RoboDK station: VUI_control.rdk

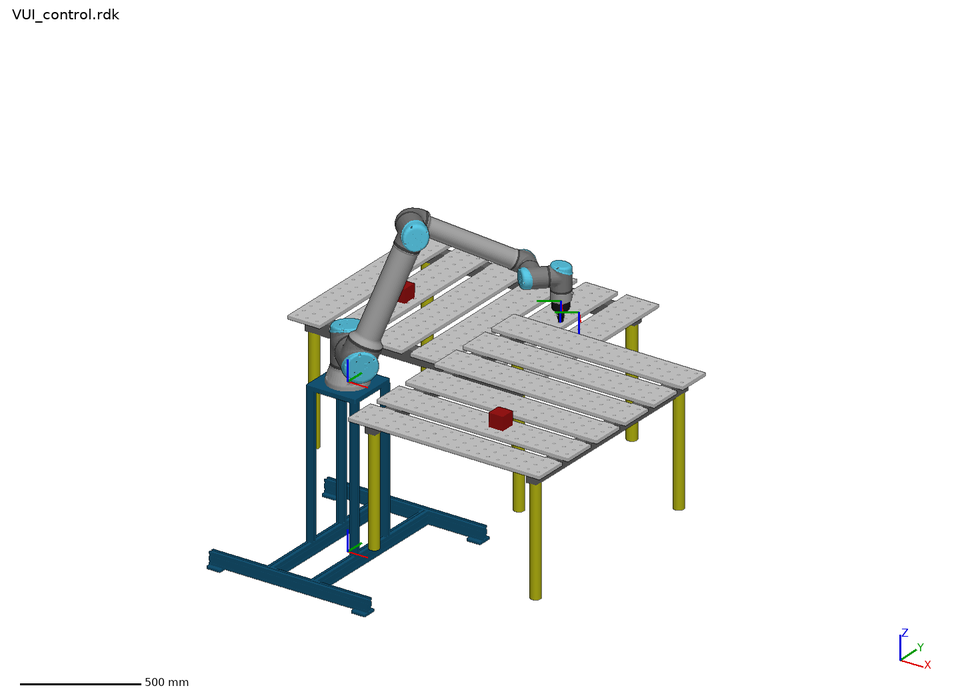
[picture v0: the station drawn from its stored meshes, robots at their saved joint values, targets as dots, program paths as lines]
Station Gripper_test (saved by RoboDK 5.3.1). Poses are relative to the parent item; angles as X-Y-Z fixed-axis rotations.
  - frame UR10e Base at (0, 0, 0) mm
    - robot UR10e: 6 axes, payload 10 kg, reach 1300 mm, repeatability 0.05 mm, weight 28.9 kg
        modified DH rows (alpha deg, a mm, theta deg, d mm): 0, 0, 0, 180.7; 90, 0, 180, 0; 0, 612.6, 0, 0; 0, 571.335, 0, 174.15; -90, 0, 0, 119.85; 90, 0, 180, 116.55
        joint limits [-360, -360, -360, -360, -360, -360] to [360, 360, 360, 360, 360, 360]; home [0, -90, -90, 0, 90, 0]; saved at [47.371, -112.765, -94.763, -63.434, 90.01, 8.604]
      - tool 2F85+FTS, TCP at (0, 0, 145) mm
      - frame RobotiQ 2F85 Base at (0, 0, 0) mm
        - robot RobotiQ 2F85: 1 axes, payload 5 kg
            joint limits [0] to [85]; home [85]; saved at [85]
        - target Open (Cartesian target) at (0, 0, 103.92) mm; joints [85] of RobotiQ 2F85
        - target Close (Cartesian target) at (0, 0, 103.92) mm; joints [3.08] of RobotiQ 2F85
        - frame ZED2i at (-64.91, -81.57, 83.4) mm
    - object Base-Robot at (0, 0, 0) mm, size 800 x 900 x 790 mm, geometry from Base-Robot.stl
  - Python program gripper_robotiq (listed below)
  - Python program main (listed below)
  - Python program UR_ActivateMonitoring (listed below)
  - frame Floor at (0, 0, -780) mm
    - object Pick_Table at (900, 0, 970) mm, rotated rx 0 ry 0 rz 90 deg, size 1193.8 x 965.2 x 609.6 mm, geometry from Object Table.wrl
      - object box at (-300, -80, 30) mm, size 71.9 x 71.9 x 71.9 mm, geometry from box.sld
    - object Place_Table at (0, 900, 750) mm, size 1193.8 x 965.2 x 609.6 mm, geometry from Object Table.wrl
      - object red at (-300, -80, 30) mm, size 71.9 x 71.9 x 71.9 mm, geometry from box.sld

--- Python program gripper_robotiq ---
"""Module to control Robotiq's grippers - tested with HAND-E"""

import socket
import threading
import time
from enum import Enum
from typing import Union, Tuple, OrderedDict


class RobotiqGripper:
    """
    Communicates with the gripper directly, via socket with string commands, leveraging string names for variables.
    """
    # WRITE VARIABLES (CAN ALSO READ)
    # act : activate (1 while activated, can be reset to clear fault status)
    ACT = 'ACT'
    # gto : go to (will perform go to with the actions set in pos, for, spe)
    GTO = 'GTO'
    ATR = 'ATR'  # atr : auto-release (emergency slow move)
    # adr : auto-release direction (open(1) or close(0) during auto-release)
    ADR = 'ADR'
    FOR = 'FOR'  # for : force (0-255)
    SPE = 'SPE'  # spe : speed (0-255)
    POS = 'POS'  # pos : position (0-255), 0 = open
    # READ VARIABLES
    STA = 'STA'  # status (0 = is reset, 1 = activating, 3 = active)
    PRE = 'PRE'  # position request (echo of last commanded position)
    # object detection (0 = moving, 1 = outer grip, 2 = inner grip, 3 = no object at rest)
    OBJ = 'OBJ'
    FLT = 'FLT'  # fault (0=ok, see manual for errors if not zero)

    ENCODING = 'UTF-8'  # ASCII and UTF-8 both seem to work

    class GripperStatus(Enum):
        """Gripper status reported by the gripper. The integer values have to match what the gripper sends."""
        RESET = 0
        ACTIVATING = 1
        # UNUSED = 2  # This value is currently not used by the gripper firmware
        ACTIVE = 3

    class ObjectStatus(Enum):
        """Object status reported by the gripper. The integer values have to match what the gripper sends."""
        MOVING = 0
        STOPPED_OUTER_OBJECT = 1
        STOPPED_INNER_OBJECT = 2
        AT_DEST = 3

    def __init__(self):
        """Constructor."""
        self.socket = None
        self.command_lock = threading.Lock()
        self._min_position = 0
        self._max_position = 255
        self._min_speed = 0
        self._max_speed = 255
        self._min_force = 0
        self._max_force = 255

    def connect(self, hostname: str, port: int, socket_timeout: float = 2.0) -> None:
        """Connects to a gripper at the given address.
        :param hostname: Hostname or ip.
        :param port: Port.
        :param socket_timeout: Timeout for blocking socket operations.
        """
        self.socket = socket.socket(socket.AF_INET, socket.SOCK_STREAM)
        self.socket.connect((hostname, port))
        self.socket.settimeout(socket_timeout)

    def disconnect(self) -> None:
        """Closes the connection with the gripper."""
        self.socket.close()

    def _set_vars(self, var_dict: OrderedDict[str, Union[int, float]]):
        """Sends the appropriate command via socket to set the value of n variables, and waits for its 'ack' response.
        :param var_dict: Dictionary of variables to set (variable_name, value).
        :return: True on successful reception of ack, false if no ack was received, indicating the set may not
        have been effective.
        """
        # construct unique command
        cmd = "SET"
        for variable, value in var_dict.items():
            cmd += f" {variable} {str(value)}"
        cmd += '\n'  # new line is required for the command to finish
        # atomic commands send/rcv
        with self.command_lock:
            self.socket.sendall(cmd.encode(self.ENCODING))
            data = self.socket.recv(1024)
        return self._is_ack(data)

    def _set_var(self, variable: str, value: Union[int, float]):
        """Sends the appropriate command via socket to set the value of a variable, and waits for its 'ack' response.
        :param variable: Variable to set.
        :param value: Value to set for the variable.
        :return: True on successful reception of ack, false if no ack was received, indicating the set may not
        have been effective.
        """
        return self._set_vars(OrderedDict([(variable, value)]))

    def _get_var(self, variable: str):
        """Sends the appropriate command to retrieve the value of a variable from the gripper, blocking until the
        response is received or the socket times out.
        :param variable: Name of the variable to retrieve.
        :return: Value of the variable as integer.
        """
        # atomic commands send/rcv
        with self.command_lock:
            cmd = f"GET {variable}\n"
            self.socket.sendall(cmd.encode(self.ENCODING))
            data = self.socket.recv(1024)

        # expect data of the form 'VAR x', where VAR is an echo of the variable name, and X the value
        # note some special variables (like FLT) may send 2 bytes, instead of an integer. We assume integer here
        var_name, value_str = data.decode(self.ENCODING).split()
        if var_name != variable:
            raise ValueError(
                f"Unexpected response {data} ({data.decode(self.ENCODING)}): does not match '{variable}'")
        value = int(value_str)
        return value

    @staticmethod
    def _is_ack(data: str):
        return data == b'ack'

    def _reset(self):
        """
        Reset the gripper.
        The following code is executed in the corresponding script function
        def rq_reset(gripper_socket="1"):
            rq_set_var("ACT", 0, gripper_socket)
            rq_set_var("ATR", 0, gripper_socket)

            while(not rq_get_var("ACT", 1, gripper_socket) == 0 or not rq_get_var("STA", 1, gripper_socket) == 0):
                rq_set_var("ACT", 0, gripper_socket)
                rq_set_var("ATR", 0, gripper_socket)
                sync()
            end

            sleep(0.5)
        end
        """
        self._set_var(self.ACT, 0)
        self._set_var(self.ATR, 0)
        while (not self._get_var(self.ACT) == 0 or not self._get_var(self.STA) == 0):
            self._set_var(self.ACT, 0)
            self._set_var(self.ATR, 0)
        time.sleep(0.5)

    def activate(self, auto_calibrate: bool = True):
        """Resets the activation flag in the gripper, and sets it back to one, clearing previous fault flags.
        :param auto_calibrate: Whether to calibrate the minimum and maximum positions based on actual motion.
        The following code is executed in the corresponding script function
        def rq_activate(gripper_socket="1"):
            if (not rq_is_gripper_activated(gripper_socket)):
                rq_reset(gripper_socket)

                while(not rq_get_var("ACT", 1, gripper_socket) == 0 or not rq_get_var("STA", 1, gripper_socket) == 0):
                    rq_reset(gripper_socket)
                    sync()
                end

                rq_set_var("ACT",1, gripper_socket)
            end
        end
        def rq_activate_and_wait(gripper_socket="1"):
            if (not rq_is_gripper_activated(gripper_socket)):
                rq_activate(gripper_socket)
                sleep(1.0)

                while(not rq_get_var("ACT", 1, gripper_socket) == 1 or not rq_get_var("STA", 1, gripper_socket) == 3):
                    sleep(0.1)
                end

                sleep(0.5)
            end
        end
        """
        if not self.is_active():
            self._reset()
            while (not self._get_var(self.ACT) == 0 or not self._get_var(self.STA) == 0):
                time.sleep(0.01)

            self._set_var(self.ACT, 1)
            time.sleep(1.0)
            while (not self._get_var(self.ACT) == 1 or not self._get_var(self.STA) == 3):
                time.sleep(0.01)

        # auto-calibrate position range if desired
        if auto_calibrate:
            self.auto_calibrate()

    def is_active(self):
        """Returns whether the gripper is active."""
        status = self._get_var(self.STA)
        return RobotiqGripper.GripperStatus(status) == RobotiqGripper.GripperStatus.ACTIVE

    def get_min_position(self) -> int:
        """Returns the minimum position the gripper can reach (open position)."""
        return self._min_position

    def get_max_position(self) -> int:
        """Returns the maximum position the gripper can reach (closed position)."""
        return self._max_position

    def get_open_position(self) -> int:
        """Returns what is considered the open position for gripper (minimum position value)."""
        return self.get_min_position()

    def get_closed_position(self) -> int:
        """Returns what is considered the closed position for gripper (maximum position value)."""
        return self.get_max_position()

    def is_open(self):
        """Returns whether the current position is considered as being fully open."""
        return self.get_current_position() <= self.get_open_position()

    def is_closed(self):
        """Returns whether the current position is considered as being fully closed."""
        return self.get_current_position() >= self.get_closed_position()

    def get_current_position(self) -> int:
        """Returns the current position as returned by the physical hardware."""
        return self._get_var(self.POS)

    def auto_calibrate(self, log: bool = True) -> None:
        """Attempts to calibrate the open and closed positions, by slowly closing and opening the gripper.
        :param log: Whether to print the results to log.
        """
        # first try to open in case we are holding an object
        (position, status) = self.move_and_wait_for_pos(
            self.get_open_position(), 64, 1)
        if RobotiqGripper.ObjectStatus(status) != RobotiqGripper.ObjectStatus.AT_DEST:
            raise RuntimeError(
                f"Calibration failed opening to start: {str(status)}")

        # try to close as far as possible, and record the number
        (position, status) = self.move_and_wait_for_pos(
            self.get_closed_position(), 64, 1)
        if RobotiqGripper.ObjectStatus(status) != RobotiqGripper.ObjectStatus.AT_DEST:
            raise RuntimeError(
                f"Calibration failed because of an object: {str(status)}")
        assert position <= self._max_position
        self._max_position = position

        # try to open as far as possible, and record the number
        (position, status) = self.move_and_wait_for_pos(
            self.get_open_position(), 64, 1)
        if RobotiqGripper.ObjectStatus(status) != RobotiqGripper.ObjectStatus.AT_DEST:
            raise RuntimeError(
                f"Calibration failed because of an object: {str(status)}")
        assert position >= self._min_position
        self._min_position = position

        if log:
            print(
                f"Gripper auto-calibrated to [{self.get_min_position()}, {self.get_max_position()}]")

    def move(self, position: int, speed: int, force: int) -> Tuple[bool, int]:
        """Sends commands to start moving towards the given position, with the specified speed and force.
        :param position: Position to move to [min_position, max_position]
        :param speed: Speed to move at [min_speed, max_speed]
        :param force: Force to use [min_force, max_force]
        :return: A tuple with a bool indicating whether the action it was successfully sent, and an integer with
        the actual position that was requested, after being adjusted to the min/max calibrated range.
        """

        def clip_val(min_val, val, max_val):
            return max(min_val, min(val, max_val))

        clip_pos = clip_val(self._min_position, position, self._max_position)
        clip_spe = clip_val(self._min_speed, speed, self._max_speed)
        clip_for = clip_val(self._min_force, force, self._max_force)

        # moves to the given position with the given speed and force
        var_dict = OrderedDict(
            [(self.POS, clip_pos), (self.SPE, clip_spe), (self.FOR, clip_for), (self.GTO, 1)])
        return self._set_vars(var_dict), clip_pos

    def move_and_wait_for_pos(self, position: int, speed: int, force: int) -> Tuple[int, ObjectStatus]:  # noqa
        """Sends commands to start moving towards the given position, with the specified speed and force, and
        then waits for the move to complete.
        :param position: Position to move to [min_position, max_position]
        :param speed: Speed to move at [min_speed, max_speed]
        :param force: Force to use [min_force, max_force]
        :return: A tuple with an integer representing the last position returned by the gripper after it notified
        that the move had completed, a status indicating how the move ended (see ObjectStatus enum for details). Note
        that it is possible that the position was not reached, if an object was detected during motion.
        """
        set_ok, cmd_pos = self.move(position, speed, force)
        if not set_ok:
            raise RuntimeError("Failed to set variables for move.")

        # wait until the gripper acknowledges that it will try to go to the requested position
        while self._get_var(self.PRE) != cmd_pos:
            time.sleep(0.001)

        # wait until not moving
        cur_obj = self._get_var(self.OBJ)
        while RobotiqGripper.ObjectStatus(cur_obj) == RobotiqGripper.ObjectStatus.MOVING:
            cur_obj = self._get_var(self.OBJ)

        # report the actual position and the object status
        final_pos = self._get_var(self.POS)
        final_obj = cur_obj
        return final_pos, RobotiqGripper.ObjectStatus(final_obj)

--- Python program main ---
try:  # 192.168.56.101
    from robodk.robolink import *
    from robodk import *
except:
    from robolink.robolink import *    # API to communicate with RoboDK
    from robodk.robodk import *      # basic matrix operations
finally:
    from AWSIoTPythonSDK.MQTTLib import AWSIoTMQTTClient
    import gripper_robotiq
    import socket
    import numpy as np
    import time
    import json
    import ast

    robot_ip = "192.168.1.10"  # Replace with your robot ip
    rdk_ip = 'localhost'  # Or the explicit ip of the computer running RoboDK
    pose = eye()

    RDK = Robolink()
    RDK.setRunMode(RUNMODE_RUN_ROBOT)  # RUNMODE_RUN_ROBOT
    robot = RDK.Item('UR10e')
    sim_gripper = RDK.Item('RobotiQ 2F85')  # the robotiq gripper inside RoboDK
    close_grp = RDK.Item("Close", ITEM_TYPE_TARGET)
    open_grp = RDK.Item("Open", ITEM_TYPE_TARGET)

    # detections=detector.GetData()

    gripper = gripper_robotiq.RobotiqGripper()
    gripper.connect(robot_ip, 63352)  # The port on the URe family is 63352
    # gripper.activate()
    gMax_Pos = gripper.get_max_position()

    clientId = "LAGID"
    host = "a1uv83ra8k1y7l-ats.iot.us-east-1.amazonaws.com"
    port = 8883
    rootCAPath = "C:/Users/LAG/Desktop/connect_device_package/root-CA.crt"
    privateKeyPath = "C:/Users/LAG/Desktop/connect_device_package/UR10_robot.private.key"
    certificatePath = "C:/Users/LAG/Desktop/connect_device_package/UR10_robot.cert.pem"
    topic_sub = "alexa/to/ur"
    topic_pub = "ur/to/alexa"
    mode = 'both'

    myAWSIoTMQTTClient = AWSIoTMQTTClient(clientId)  # ,useWebsocket=True)
    myAWSIoTMQTTClient.configureEndpoint(host, port)
    myAWSIoTMQTTClient.configureCredentials(
        rootCAPath, privateKeyPath, certificatePath)

    myAWSIoTMQTTClient.configureAutoReconnectBackoffTime(1, 32, 20)
    myAWSIoTMQTTClient.configureOfflinePublishQueueing(-1)
    myAWSIoTMQTTClient.configureDrainingFrequency(2)  # Draining: 2 Hz
    myAWSIoTMQTTClient.configureConnectDisconnectTimeout(10)  # 10 sec
    myAWSIoTMQTTClient.configureMQTTOperationTimeout(5)  # 5 sec
    myAWSIoTMQTTClient.connect()

    client_socket = socket.socket(socket.AF_INET, socket.SOCK_STREAM)
    host_ip = "10.25.147.84"
    port = 50007
    client_socket.connect((host_ip, port))

    # Global variables
    command_action = 0
    extra_value = 0
    name_save = ""
    current_prog = ""
    flag_create = False
    flag_frame = True
    flag_firstpoint = True
    gripper_status = True
    save_value = 0
    save_name = ""
    pick_flag = False
    place_flag = False

    state_record = 0
    speed = 150
    force = 20

    place_zone = [270, -90, 90, -90, -90, 0, False]
    pick_zone = [0, -90, -90, -90, 90, 0, True]

    class State(dict):
        def __setitem__(self, name, value):
            super().__setitem__(name, value)

    class Program:
        def __init__(self, home, frame, states):
            self.home = home
            self.frame = frame
            self.states = states

    def log_info(gripper):
        print(f"Pos: {str(gripper.get_current_position()): >3} "
              f"Open: {gripper.is_open(): <2} "
              f"Closed: {gripper.is_closed(): <2} ")

    def dt_gripper_position(current_position):
        dt_pos = [0]
        dt_pos[0] = 85 - (current_position / gMax_Pos) * 85
        return dt_pos

    def open_gripper():
        if RDK.RunMode() > 1:
            RDK.setRunMode(1)
        time.sleep(0.5)
        gripper.move_and_wait_for_pos(0, 255, 255)
        log_info(gripper)
        dt_pos = dt_gripper_position(gripper.get_current_position())
        sim_gripper.MoveJ(dt_pos)
        time.sleep(0.5)
        # tool_frame.DetachAll()
        RDK.setRunMode(6)
        time.sleep(0.5)

    def close_gripper():
        if RDK.RunMode() > 1:
            RDK.setRunMode(1)
        gripper.move_and_wait_for_pos(int(gMax_Pos/2), 255, 191)
        log_info(gripper)
        dt_pos = dt_gripper_position(gripper.get_current_position())
        sim_gripper.MoveJ(dt_pos)
        #input("Press 'Enter' to continue...")
        gripper.move_and_wait_for_pos(gMax_Pos, 255, 191)
        log_info(gripper)
        dt_pos = dt_gripper_position(gripper.get_current_position())
        sim_gripper.MoveJ(dt_pos)
        #input("Press 'Enter' to continue...")
        time.sleep(0.5)
        # tool_frame.AttachClosest()
        RDK.setRunMode(6)
        time.sleep(0.5)

    def publishMqtt(alert):
        # print("publishsing...")
        mess = {}
        mess["value"] = "mqtt"
        mess['message'] = alert
        messageJson = json.dumps(mess)
        myAWSIoTMQTTClient.publish(topic_pub, messageJson, 1)
        return 0

    def controlRobot(target):  # change when run or simulate
        global gripper_status
        if isinstance(target, list):
            robot.MoveJ(target)
            if target[6] == True:
                # sim_gripper.MoveJ(open_grp)
                gripper.move_and_wait_for_pos(5, speed, force)
                gripper_status = True
            else:
                # sim_gripper.MoveJ(close_grp)
                gripper.move_and_wait_for_pos(200, speed, force)
                gripper_status = False
        elif isinstance(target, dict):
            c = target.popitem()
            count = int(c[1])
            while count != 0:
                keys_list = [*target]  # list(target.keys())
                for key in keys_list:
                    robot.MoveJ(target[key])
                    if target[key][6] == True:
                        # sim_gripper.MoveJ(open_grp)
                        gripper.move_and_wait_for_pos(5, speed, force)
                    else:
                        # sim_gripper.MoveJ(close_grp)
                        gripper.move_and_wait_for_pos(200, speed, force)
                count -= 1
        elif target:
            gripper.move_and_wait_for_pos(target, speed, force)
            # sim_gripper.MoveJ(target)

        else:
            return 0

    def createProg(prog_name):
        with open("C:/Users/LAG/Documents/RoboDK/savedprog_data.json", "r") as jsonFile:
            savedPrograms = json.load(jsonFile)
        if prog_name in savedPrograms:
            return "A program with that name already exists, do you want to edit it? or try another name"
        else:
            global flag_create
            global current_prog
            flag_create = True
            prog = Program(None, None, State())
            savedPrograms[prog_name] = prog.__dict__
            with open("C:/Users/LAG/Documents/RoboDK/savedprog_data.json", "w") as jsonFile:
                json.dump(savedPrograms, jsonFile)
            jsonFile.close()
            current_prog = prog_name
            return f"{prog_name} was created succesfully"

    def selectFrame(frame):
        global flag_frame

        if flag_create == True or current_prog:
            with open('default_data.json', "r") as jsonFile:
                data = json.load(jsonFile)
                frame = data["frames"][frame]
            jsonFile.close()
            with open("C:/Users/LAG/Documents/RoboDK/savedprog_data.json", "r") as jsonFile:
                savedPrograms = json.load(jsonFile)
                savedPrograms[current_prog]["frame"] = frame
            with open("C:/Users/LAG/Documents/RoboDK/savedprog_data.json", "w") as jsonFile:
                json.dump(savedPrograms, jsonFile)
            jsonFile.close()
            flag_frame = True
            return "Frame saved succesfully"
        else:
            return "I need a program name"

    def selectFirstPoint(first_point):
        global flag_firstpoint
        if flag_create == True and flag_frame == True or current_prog:
            with open('default_data.json', "r") as jsonFile:
                data = json.load(jsonFile)
                first_point = data["homes"][first_point]
            jsonFile.close()
            with open("C:/Users/LAG/Documents/RoboDK/savedprog_data.json", "r") as jsonFile:
                savedPrograms = json.load(jsonFile)
                savedPrograms[current_prog]["home"] = first_point
            with open("C:/Users/LAG/Documents/RoboDK/savedprog_data.json", "w") as jsonFile:
                json.dump(savedPrograms, jsonFile)
            jsonFile.close()
            flag_firstpoint = True
            return "First point saved succesfully"
        else:
            return "I need a program name"

    def saveState(val, state_name):

        global state_record, pick_zone, place_zone
        joints = []
        auxjoint = tr(robot.Joints())
        for item in auxjoint:
            joints.append(item[0])
        joints.append(gripper_status)

        if int(val) != 0:
            if int(val) == 1:
                pick_zone = joints
                print(pick_zone)
                return " pick Zone saved"
            else:
                place_zone = joints
                return " place Zone saved"

        else:
            if state_name:
                savedStates = State()
                savedStates[state_name] = joints
                with open("C:/Users/LAG/Documents/RoboDK/savedprog_data.json", "r") as jsonFile:
                    savedPrograms = json.load(jsonFile)
                    savedPrograms[current_prog]["states"][state_name] = joints
                with open("C:/Users/LAG/Documents/RoboDK/savedprog_data.json", "w") as jsonFile:
                    json.dump(savedPrograms, jsonFile)
                jsonFile.close()
                return "Saved state"
            else:
                state_record = state_record+1
                state_num = str(state_record)
                savedStates = State()
                savedStates[state_num] = joints
                with open("C:/Users/LAG/Documents/RoboDK/savedprog_data.json", "r") as jsonFile:
                    savedPrograms = json.load(jsonFile)
                    savedPrograms[current_prog]["states"][state_num] = joints
                with open("C:/Users/LAG/Documents/RoboDK/savedprog_data.json", "w") as jsonFile:
                    json.dump(savedPrograms, jsonFile)
                jsonFile.close()
                return "Saved state"

    def programingMode(val, state_name):
        if flag_firstpoint == True and flag_frame == True and current_prog:
            return saveState(val, state_name)
        else:
            return "I understand, you want to save this pose, but in which program? Create or edit a program"

    def getPoint(state_name):
        with open("C:/Users/LAG/Documents/RoboDK/savedprog_data.json", "r") as jsonFile:
            savedPrograms = json.load(jsonFile)
            print(state_name)
            target = savedPrograms[current_prog]["states"][f"point {state_name}"]
        return target

    def controlGripper(action):  # change when run or simulate
        global gripper_status

        if action == 0 and gripper_status == True:
            gripper_status = False
            return "Closing gripper", 200  # close_grp
        elif action == 0 and gripper_status == False:
            return "Gripper is already closed", None
        elif action == 1 and gripper_status == False:
            gripper_status = True
            return "Opening gripper", 5  # open_grp
        elif action == 1 and gripper_status == True:
            return "Gripper is already opened", None
        elif action == 2 and gripper_status == False:
            gripper_status = True
            return "Opening gripper", 5  # open_grp
        elif action == 2 and gripper_status == True:
            gripper_status = False
            return "Closing gripper", 200  # close_grp

    def controlMove(comm_a, pointname):
        global gripper_status
        target = []
        action, unit, num = int(comm_a[0]), int(comm_a[1]), int(comm_a[2:])
        if unit == 0:
            val_move = num
        else:
            val_move = num*10
        if action == 0:
            target = [0, -90, 0, 0, 90, 0, True]
            msn = "moving home"
            return msn, target
        if action == 1:
            current_pose = robot.Pose()
            new_pose = current_pose.Offset(0, val_move, 0)
            new_joints = robot.SolveIK(new_pose, tool=robot.PoseTool())
            if len(new_joints.tolist()) < 6:
                msn = "No robot solution!! The new position is too far, out of reach or close to a singularity"
            else:
                msn = "moving right"
                target = new_joints.tolist()
                target.append(gripper_status)
            return msn, target
        if action == 2:
            current_pose = robot.Pose()
            new_pose = current_pose.Offset(0, -val_move, 0)
            new_joints = robot.SolveIK(new_pose, tool=robot.PoseTool())
            if len(new_joints.tolist()) < 6:
                msn = "No robot solution!! The new position is too far, out of reach or close to a singularity"
            else:
                msn = "moving left"
                target = new_joints.tolist()
                target.append(gripper_status)
            return msn, target
        if action == 3:
            current_pose = robot.Pose()
            new_pose = current_pose.Offset(0, 0, val_move)
            new_joints = robot.SolveIK(new_pose, tool=robot.PoseTool())
            if len(new_joints.tolist()) < 6:
                msn = "No robot solution!! The new position is too far, out of reach or close to a singularity"
            else:
                msn = "moving up"
                target = new_joints.tolist()
                target.append(gripper_status)
            return msn, target
        if action == 4:
            current_pose = robot.Pose()
            new_pose = current_pose.Offset(0, 0, -val_move)
            new_joints = robot.SolveIK(new_pose, tool=robot.PoseTool())
            if len(new_joints.tolist()) < 6:
                msn = "No robot solution!! The new position is too far, out of reach or close to a singularity"
            else:
                msn = "moving down"
                target = new_joints.tolist()
                target.append(gripper_status)
            return msn, target
        if action == 5:
            current_pose = robot.Pose()
            new_pose = current_pose.Offset(val_move, 0, 0)
            new_joints = robot.SolveIK(new_pose, tool=robot.PoseTool())
            if len(new_joints.tolist()) < 6:
                msn = "No robot solution!! The new position is too far, out of reach or close to a singularity"
            else:
                msn = "moving forward"
                target = new_joints.tolist()
                target.append(gripper_status)
            return msn, target
        if action == 6:
            current_pose = robot.Pose()
            new_pose = current_pose.Offset(-val_move, 0, 0)
            new_joints = robot.SolveIK(new_pose, tool=robot.PoseTool())
            if len(new_joints.tolist()) < 6:
                msn = "No robot solution!! The new position is too far, out of reach or close to a singularity"
            else:
                msn = "moving backwards"
                target = new_joints.tolist()
                target.append(gripper_status)
            return msn, target
        if action == 7:
            target = getPoint(pointname)
            msn = f"moving to point {pointname}, send from py"
            return msn, target

    def controlRotate(values):

        target = []
        axis, direction = int(values[0]), int(values[1])

        if axis == 0:
            current_pose = robot.Pose()
            if direction == 1:
                new_pose = current_pose.RelTool(0, 0, 0, rx=36)
            else:
                new_pose = current_pose.RelTool(0, 0, 0, rx=-36)
            new_joints = robot.SolveIK(new_pose, tool=robot.PoseTool())
            if len(new_joints.tolist()) < 6:
                msn = "No robot solution!! The new position is too far, out of reach or close to a singularity"
            else:
                msn = "rotating in x axis"
                target = new_joints.tolist()
                target.append(gripper_status)
            return msn, target
        if axis == 1:
            current_pose = robot.Pose()
            if direction == 1:
                new_pose = current_pose.RelTool(0, 0, 0, ry=36)
            else:
                new_pose = current_pose.RelTool(0, 0, 0, ry=-36)
            new_joints = robot.SolveIK(new_pose, tool=robot.PoseTool())
            if len(new_joints.tolist()) < 6:
                msn = "No robot solution!! The new position is too far, out of reach or close to a singularity"
            else:
                msn = "rotating in y axis"
                target = new_joints.tolist()
                target.append(gripper_status)
            return msn, target
        if axis == 2:
            current_pose = robot.Pose()
            if direction == 1:
                new_pose = current_pose.RelTool(0, 0, 0, rz=-36)
            else:
                new_pose = current_pose.RelTool(0, 0, 0, rz=36)
            new_joints = robot.SolveIK(new_pose, tool=robot.PoseTool())
            if len(new_joints.tolist()) < 6:
                msn = "No robot solution!! The new position is too far, out of reach or close to a singularity"
            else:
                msn = "rotating in z axis"
                target = new_joints.tolist()
                target.append(gripper_status)
            return msn, target

    def runningMode(running_program, counter):
        with open("C:/Users/LAG/Documents/RoboDK/savedprog_data.json", "r") as jsonFile:
            savedPrograms = json.load(jsonFile)
        if running_program in savedPrograms:
            states = savedPrograms[running_program]["states"]
            states.update({"count": counter})
            msn = f"Running {running_program}"
            return msn, states
        else:
            return "Invalid program name, try with other name or ask for the list", None

    def getDatajetson(selec):
        time.sleep(1)
        client_socket.send(b"Data")
        answ_byte = client_socket.recv(1024).decode()
        answ_dict = ast.literal_eval(answ_byte)
        if selec == 0:
            try:
                return answ_dict[save_value]
            except:
                time.sleep(1)
                client_socket.send(b"Data")
                answ_byte = client_socket.recv(1024).decode()
                answ_dict = ast.literal_eval(answ_byte)
                return answ_dict[save_value]
        else:
            try:
                return answ_dict[save_name]
            except:
                time.sleep(1)
                client_socket.send(b"Data")
                answ_byte = client_socket.recv(1024).decode()
                answ_dict = ast.literal_eval(answ_byte)
                return answ_dict[save_name]

    def logicRobot(command, name, value):
        global command_action, name_save, extra_value, save_value, save_name, pick_flag, place_flag
        target = []

        if pick_flag == True:
            while robot.Busy() == 1:
                time.sleep(1)
            msg = ""
            for i in range(2):
                coord = getDatajetson(0)
            base = robot.Pose()
            zed_pose = Pose(coord[0], coord[1], coord[2], -0, 0, 0)
            tool_pose = zed_pose*transl(-64.91, -81.570, -61.6)
            new_robot_position = base*tool_pose
            new_robot_joints = robot.SolveIK(
                pose=new_robot_position, tool=Pose(0, 0, 145, 0, 0, 0))
            target = new_robot_joints.tolist()
            target.append(False)
            pick_flag = False
            flag = True

        elif place_flag == True:
            while robot.Busy() == 1:
                time.sleep(1)
            msg = ""
            coord = getDatajetson(2)
            base = robot.Pose()
            zed_pose = Pose(coord[0], coord[1], coord[2], -0, 0, 0)
            tool_pose = zed_pose*transl(-64.91, -81.570, -61.6)
            new_robot_position = base*tool_pose
            new_robot_joints = robot.SolveIK(
                pose=new_robot_position, tool=Pose(0, 0, 145, 0, 0, 0))
            #target = new_robot_joints.tolist()
            if save_name == "green":
                target = [91.14, -128, -101, -38, 90, 0]
            else:
                target = [110, -128, -102, -40, 90, 20]
            target.append(True)
            place_flag = False
            flag = True

        else:

            if command == 1:  # move command
                res = controlMove(value, name)
                msg = res[0]
                target = res[1]
                flag = True
            elif command == 2:  # gripper control
                res = controlGripper(value)
                msg = res[0]
                target = res[1]
                flag = True
            elif command == 3:  # create program
                msg = createProg(name)
                flag = True
            elif command == 4:  # select Frame
                msg = selectFrame(name)
                flag = True
            elif command == 5:  # select point 0
                msg = selectFirstPoint(name)
                flag = True
            elif command == 6:  # save state
                msg = programingMode(value, name)
                flag = True
            elif command == 7:  # run programs
                res = runningMode(name, value)
                msg = res[0]
                target = res[1]
                flag = True
            elif command == 8:  # pick
                msg = "Ok, Im searching the part"
                target = pick_zone
                save_value = value
                pick_flag = True
                flag = True
            elif command == 9:  # place
                msg = "Perfect, Im searching the zone"
                target = place_zone
                save_name = name
                place_flag = True
                flag = True
            elif command == 10:  # rotate
                res = controlRotate(value)
                msg = res[0]
                target = res[1]
                flag = True
            else:
                # print("subscribe...")
                return 0

        if flag == True:
            if msg:
                publishMqtt(msg)
            if target:
                controlRobot(target)

        flag = False
        command_action = 0
        name_save = ""
        extra_value = 0

    def customCallback(self, userdata, message):
        global command_action
        global name_save
        global extra_value
        data = json.loads(message.payload)
        command_action = data["command"]
        extra_value = data["value"]
        name_save = data["name"]

    def subs():
        myAWSIoTMQTTClient.subscribe(topic_sub, 1, customCallback)

    success = robot.Connect()
    status, status_msg = robot.ConnectedState()

    if status != ROBOTCOM_READY:
        # Stop if the connection did not succeed
        print(status_msg)
        raise Exception("Failed to connect: " + status_msg)

    if __name__ == "__main__":
        while True:
            subs()
            logicRobot(command_action, name_save, extra_value)
            time.sleep(0.5)  # 1

--- Python program UR_ActivateMonitoring ---
# This script creates a thread to monitor the position and other variables from a real UR robot
# With this script active, RoboDK will create a new target when the robot is moved a certain tolerance
#
# More information about the RoboDK API here:
# https://robodk.com/doc/en/RoboDK-API.html
# Press F5 to run the script
# Or visit: https://robodk.com/doc/en/PythonAPI/index.html
from robolink import *    # API to communicate with RoboDK
from robodk import *      # basic matrix operations
import threading
import socket
import struct
import os
import time

# Refresh the screen every time the robot position changes
TOLERANCE_JOINTS_REFRESH   = 0.1
RETRIEVE_JOINTS_ONCE = False  # If True, the current robot position will be retrieved once only

# Create targets given a tolerance in degrees
CREATE_TARGETS = False
TOLERANCE_JOINTS_NEWTARGET = 10 # in degrees

REFRESH_RATE = 0.01

# Make current robot joints accessible in case we run it on a separate thread
global ROBOT_JOINTS


# Procedure to check if robot joint positions are different according to a certain tolerance
def Robot_Joints_Check(jA,jB, tolerance_deg=1):
    if jA is None:
        return True

    for i in range(6):
        if abs(jA[i]-jB[i]) > tolerance_deg*pi/180:
            return True
    return False

#########################################################################
# Byte shifts to point to the right byte data inside a packet
UR_GET_TIME = 1
UR_GET_JOINT_POSITIONS = 252
UR_GET_JOINT_SPEEDS = 300
UR_GET_JOINT_CURRENTS = 348
UR_GET_TCP_FORCES = 540

# Get packet size according to the byte array
def packet_size(buf):
    if len(buf) < 4:
        return 0
    return struct.unpack_from("!i", buf, 0)[0]

# Check if a packet is complete
def packet_check(buf):
    msg_sz = packet_size(buf)
    if len(buf) < msg_sz:
        print("Incorrect packet size %i vs %i" % (msg_sz, len(buf)))
        return False

    return True

# Get specific information from a packet
def packet_value(buf, offset, nval=6):
    if len(buf) < offset+nval:
        print("Not available offset (maybe older Polyscope version?): %i - %i" % (len(buf), offset))
        return None
    format = '!'
    for i in range(nval):
        format+='d'
    return list(struct.unpack_from(format, buf, offset))    #return list(struct.unpack_from("!dddddd", buf, offset))

# Action to take when a new packet arrives
def on_packet(packet):
    global ROBOT_JOINTS
    # Retrieve desired information from a packet
    rob_joints_RAD = packet_value(packet, UR_GET_JOINT_POSITIONS)
    ROBOT_JOINTS = [ji * 180.0/pi for ji in rob_joints_RAD]
    #ROBOT_SPEED = packet_value(packet, UR_GET_JOINT_SPEEDS)
    #ROBOT_CURRENT = packet_value(packet, UR_GET_JOINT_CURRENTS)
    #print(ROBOT_JOINTS)

# Monitor thread to retrieve information from the robot
def UR_Monitor():
    while True:
        rt_socket = socket.create_connection((ROBOT_IP, ROBOT_PORT))
        buf = b''
        packet_count = 0
        packet_time_last = time.time()
        while True:
            more = rt_socket.recv(4096)
            if more:
                buf = buf + more
                if packet_check(buf):
                    packet_len = packet_size(buf)
                    packet, buf = buf[:packet_len], buf[packet_len:]
                    on_packet(packet)
                    packet_count += 1
                    if packet_count % 125 == 0:
                        t_now = time.time()
                        print("Monitoring at %.1f packets per second" % (packet_count/(t_now-packet_time_last)))
                        packet_count = 0
                        packet_time_last = t_now

        rt_socket.close()
#########################################################################

# Enter RoboDK IP and Port
ROBOT_IP = None #'192.168.2.31'
ROBOT_PORT = 30003

# Start RoboDK API
RDK = Robolink()

# Retrieve a robot
robot = RDK.ItemUserPick('Select a UR robot to retrieve current position', ITEM_TYPE_ROBOT)
if not robot.Valid():
    quit()

# Retrieve Robot's IP:
if ROBOT_IP is None:
    ip,port,path,ftpuser,ftppass = robot.ConnectionParams()
    ROBOT_IP = ip



ROBOT_JOINTS = None
last_joints_target = None
last_joints_refresh = None

# Start the Robot Monitor thread
#q = queue.Queue()
t = threading.Thread(target=UR_Monitor)
t.daemon = True
t.start()
#UR_Monitor()

# Start the main loop to refresh RoboDK and create targets/programs automatically
target_count = 0
while True:
    # Wait for a valid robot joints reading
    if ROBOT_JOINTS is None:
        continue

    # Set the robot to that position
    if Robot_Joints_Check(last_joints_refresh, ROBOT_JOINTS, TOLERANCE_JOINTS_REFRESH):
        last_joints_refresh = ROBOT_JOINTS
        robot.setJoints(ROBOT_JOINTS)

    # Stop here if we need only the current position
    if RETRIEVE_JOINTS_ONCE:
        quit(0)

    # Check if the robot has moved enough to create a new target
    if CREATE_TARGETS and Robot_Joints_Check(last_joints_target, ROBOT_JOINTS, TOLERANCE_JOINTS_NEWTARGET):
        last_joints_target = ROBOT_JOINTS
        target_count = target_count + 1
        newtarget = RDK.AddTarget('T %i' % target_count, 0, robot)

    # Take a short break
    pause(REFRESH_RATE)
